{attribute 'c++_compatible'}
FUNCTION_BLOCK MruInterface IMPLEMENTS ITcIoUdpProtocolRecv
VAR_INPUT
	
END_VAR
VAR_OUTPUT
	feedback			: FeedbackMru;
END_VAR
VAR	
	// UDP connection
	{attribute 'TcInitSymbol'}
	oid					: OTCID;
	ipUdp 				: ITcIoUdpProtocol;
	recvCounter			: UDINT := 0;
	localUdpPort		: UINT;
	
	// UDP raw data structures
	rxUdpDataBE			: RxMru;	// Big endian data struct
	rxUdpData			: RxMru;	// Host/little endian data struct
	
	// HMI data
	pTxHmiData			: PVOID;
	txHmiData			: TxHmiMru;
END_VAR

// Update IO data
UpdateIO();

// Update UDP data
UpdateUDP();

// Update HMI data
UpdateHMI();

METHOD BigToLittleEndian : REAL
VAR_INPUT
	realIn		: REAL;
END_VAR

VAR
	realOut		: REAL;	

	bytesIn		: ARRAY [0..3] OF BYTE;
	bytesOut	: ARRAY [0..3] OF BYTE;
END_VAR
// Copy to byte array
MEMCPY(ADR(bytesIn), ADR(realIn), 4);

// Switch bytes
bytesOut[3] := bytesIn[0];
bytesOut[2] := bytesIn[1];
bytesOut[1] := bytesIn[2];
bytesOut[0] := bytesIn[3];

// Copy switched butes to realOut
MEMCPY(ADR(realOut), ADR(bytesOut), 4);

// Return switched version of realIn
BigToLittleEndian := realOut;
END_METHOD

METHOD FB_exit : BOOL
VAR_INPUT
	bInCopyCode : BOOL; // if TRUE, the exit method is called for exiting an instance that is copied afterwards (online change).
END_VAR
IF (NOT bInCopyCode AND ipUdp <> 0) THEN //Shutdown
	ipUdp.UnregisterReceiver(localUdpPort);
	FW_SafeRelease(ADR(ipUdp));
	FB_exit := TRUE;
ELSE
	FB_exit := FALSE;
END_IF
END_METHOD

METHOD FB_init : BOOL
VAR_INPUT
	bInitRetains 		: BOOL; // if TRUE, the retain variables are initialized (warm start / cold start)
	bInCopyCode 		: BOOL;  // if TRUE, the instance afterwards gets moved into the copy code (online change)
	
	// Contructor arguments
	_localUdpPort 		: UINT;
	_pTxHmiData			: PVOID;
END_VAR

VAR
	ipSrv				: ITComObjectServer;
	hr 					: HRESULT;
END_VAR
// Initilize parameters
localUdpPort := _localUdpPort;
pTxHmiData := _pTxHmiData;

IF NOT bInCopyCode THEN // no online change
	IF ipUdp = 0 THEN
	    hr := FW_ObjMgr_GetObjectInstance(oid:=oid, iid:=TC_GLOBAL_IID_LIST.IID_ITcIoUdpProtocol, pipUnk:=ADR(ipUdp) );
		
		IF (SUCCEEDED(hr) AND ipUdp.RegisterReceiver(localUdpPort, THIS^) = 0 ) THEN //open local port
			FB_init := TRUE;
		ELSE
			FB_init := FALSE;			
			FW_SafeRelease(ADR(ipUdp));
		END_IF				
	END_IF
END_IF
END_METHOD

METHOD FB_reinit : BOOL
VAR_INPUT
END_VAR
IF (ipUdp <> 0) THEN 
	ipUdp.RegisterReceiver(localUdpPort, THIS^);
END_IF
END_METHOD

{attribute 'c++_compatible'}
{attribute 'signature_flag' := '33554688'}
{attribute 'pack_mode' := '1'}
{attribute 'show'}
{attribute 'minimal_input_size' := '4'}
{attribute 'checksuperglobal'}
METHOD ReceiveData : HRESULT
VAR_INPUT
	ipAddr			: UDINT;
	udpDestPort		: UINT;
	udpSrcPort		: UINT;
	nData			: UDINT;
	pData			: PVOID;
	pVlan			: POINTER TO ETYPE_VLAN_HEADER := 0;
END_VAR
// Send and receive data if the received data size is correct
IF (nData = SIZEOF(RxMru)) THEN
	// Count number of recieved UDP packets
	recvCounter := recvCounter + 1;

	// Copy data to recv buffer
	MEMCPY(ADR(rxUdpDataBE), pData, nData);
END_IF
END_METHOD

{attribute 'c++_compatible'}
{attribute 'signature_flag' := '33554688'}
{attribute 'pack_mode' := '1'}
{attribute 'show'}
{attribute 'minimal_input_size' := '4'}
{attribute 'checksuperglobal'}
METHOD TcAddRef : UDINT
END_METHOD

{attribute 'c++_compatible'}
{attribute 'signature_flag' := '33554688'}
{attribute 'pack_mode' := '1'}
{attribute 'show'}
{attribute 'minimal_input_size' := '4'}
{attribute 'checksuperglobal'}
METHOD TcQueryInterface : HRESULT
VAR_INPUT
	iid	: REFERENCE TO IID;
	pipItf	: POINTER TO PVOID;
END_VAR
END_METHOD

{attribute 'c++_compatible'}
{attribute 'signature_flag' := '33554688'}
{attribute 'pack_mode' := '1'}
{attribute 'show'}
{attribute 'minimal_input_size' := '4'}
{attribute 'checksuperglobal'}
METHOD TcRelease : UDINT
END_METHOD

METHOD PRIVATE UpdateHMI : BOOL
VAR_INPUT
END_VAR
txHmiData.status := -1;


// Update global HMI data
MEMCPY(pTxHmiData, ADR(txHmiData), SIZEOF(txHmiData));
END_METHOD

METHOD PRIVATE UpdateIO : BOOL
VAR_INPUT
END_VAR
// Update feedback data
feedback.heave := rxUdpData.PosMru_D;
feedback.heave_t := rxUdpData.VelMru_D;
feedback.heave_tt := rxUdpData.AccMru_D;
feedback.turn_rate := rxUdpData.AngRate_D;
feedback.phi := rxUdpData.Roll;
feedback.theta := rxUdpData.Pitch;
feedback.psi := rxUdpData.Yaw;
feedback.wx := rxUdpData.AngRate_R;
feedback.wy := rxUdpData.AngRate_P;
feedback.wz := rxUdpData.AngRate_Y;
feedback.wx_t := rxUdpData.AngAcc_R;
feedback.wy_t := rxUdpData.AngAcc_P;
feedback.wz_t := rxUdpData.AngAcc_Y;
feedback.x_t := rxUdpData.VelMru_R;
feedback.y_t := rxUdpData.VelMru_P;
feedback.z_t := rxUdpData.VelMru_Y;
feedback.x_tt := rxUdpData.AccMru_R;
feedback.y_tt := rxUdpData.AccMru_P;
feedback.z_tt := rxUdpData.AccMru_Y;
END_METHOD

METHOD PRIVATE UpdateUDP : BOOL
VAR_INPUT
END_VAR
// Check for incoming UDP data
IF ipUdp <> 0 THEN
	ipUdp.CheckReceived();
END_IF

// TODO: Fix this ina  more elegant way
rxUdpData.mruOK := rxUdpDataBE.mruOK;
rxUdpData.dataLength := rxUdpDataBE.dataLength;
rxUdpData.token := rxUdpDataBE.token;
rxUdpData.checksum := rxUdpDataBE.checksum;

// Big to little endian real data conversion
rxUdpData.Temperature := BigToLittleEndian(rxUdpDataBE.Temperature);
rxUdpData.PosMru_D := BigToLittleEndian(rxUdpDataBE.PosMru_D);
rxUdpData.VelMru_D := BigToLittleEndian(rxUdpDataBE.VelMru_D);
rxUdpData.AccMru_D := BigToLittleEndian(rxUdpDataBE.AccMru_D);
rxUdpData.AngRate_D := BigToLittleEndian(rxUdpDataBE.AngRate_D);
rxUdpData.Roll := BigToLittleEndian(rxUdpDataBE.Roll);
rxUdpData.Pitch := BigToLittleEndian(rxUdpDataBE.Pitch);
rxUdpData.Yaw := BigToLittleEndian(rxUdpDataBE.Yaw);
rxUdpData.AngRate_R := BigToLittleEndian(rxUdpDataBE.AngRate_R);
rxUdpData.AngRate_P := BigToLittleEndian(rxUdpDataBE.AngRate_P);
rxUdpData.AngRate_Y := BigToLittleEndian(rxUdpDataBE.AngRate_Y);
rxUdpData.AngAcc_R := BigToLittleEndian(rxUdpDataBE.AngAcc_R);
rxUdpData.AngAcc_P := BigToLittleEndian(rxUdpDataBE.AngAcc_P);
rxUdpData.AngAcc_Y := BigToLittleEndian(rxUdpDataBE.AngAcc_Y);
rxUdpData.VelMru_R := BigToLittleEndian(rxUdpDataBE.VelMru_R);
rxUdpData.VelMru_P := BigToLittleEndian(rxUdpDataBE.VelMru_P);
rxUdpData.VelMru_Y := BigToLittleEndian(rxUdpDataBE.VelMru_Y);
rxUdpData.AccMru_R := BigToLittleEndian(rxUdpDataBE.AccMru_R);
rxUdpData.AccMru_P := BigToLittleEndian(rxUdpDataBE.AccMru_P);
rxUdpData.AccMru_Y := BigToLittleEndian(rxUdpDataBE.AccMru_Y);
END_METHOD

END_FUNCTION_BLOCK

(* stored: Version 1.1.0.1, ProductVersion 3.1.4020.12
   POU MruInterface: Id {37c28233-65ff-4bfc-a679-1cd8072f7c6a}, SpecialFunc None
   Method BigToLittleEndian: Id {416b707d-216b-4813-9456-5553fa3d442d}
   Method FB_exit: Id {394f0e07-dc6c-4427-80e5-29affa6a0a68}
   Method FB_init: Id {5eb1cd80-1484-4464-b0ac-719d03818352}
   Method FB_reinit: Id {5e5db883-8291-461e-9ca2-4bf5ac87bbdf}
   Method ReceiveData: Id {46c77509-ed4e-493b-b135-d23950772b1d}
   Method TcAddRef: Id {8ef63c0d-b1c2-4674-91a1-6da67289f9a3}
   Method TcQueryInterface: Id {7c72fab3-d1fe-4b3f-b506-2e849de0d9a5}
   Method TcRelease: Id {4af70886-7416-4bc3-9a08-7cd45e097ccb}
   Method UpdateHMI: Id {f8f2096c-5401-4415-a0c4-0a80abb13107}
   Method UpdateIO: Id {041d36bb-aa8d-418e-bebf-d23d40bbfb46}
   Method UpdateUDP: Id {9d658cbb-018f-4254-bf3c-3f962c07dc24} *)
